Fanuc KAREL source: ks00049.KL

-- PROVISIONAL review KL for V770-1; original PC SHA256 45bcbc9a3b139616c803c9329d51e9163a9a66cae3eb7a3f011b941c1f7f63b5
-- Incomplete behavior may be omitted. Consult companion uncertainty JSON. Do not deploy.
PROGRAM KS00049
%NOLOCKGROUP
BEGIN
  -- UNRESOLVED_PC offsets 5-13; opcodes 3F,75
  -- UNRESOLVED_PC offsets 18-27; opcodes 3F,75
  -- UNRESOLVED_PC offsets 32-70; opcodes 27,22,22,2A,22,2A,22,22,B0
  -- UNRESOLVED_PC offsets 75-79; opcodes 7F
END KS00049
